(* IEC 61131-3 sources: ATCMcontrol_Engineering/src/TargetBase/Libs/ATCM_XMLfile, 11 files *)

(* ---- XMLClose.st ---- *)
(*[[
    UserURL="ATCMfile:XMLClose.htm",
]]*)
FUNCTION XMLClose:DWORD
VAR_INPUT
    XMLhandle : DINT;
END_VAR

inline { STDLIB(XMLClose) }

END_FUNCTION

(* ---- XMLOpen.st ---- *)
(*[[
    UserURL="ATCMfile:XMLOpen.htm",
]]*)
FUNCTION XMLOpen:DWORD
VAR_INPUT
    path : STRING;
    mode : WORD;
END_VAR
VAR_OUTPUT
    XMLhandle : DINT;
END_VAR

inline { STDLIB(XMLOpen) }

END_FUNCTION

(* ---- XMLRead.st ---- *)
(*[[
    UserURL="ATCMfile:XMLRead.htm",
]]*)
FUNCTION XMLRead:DWORD
VAR_INPUT
    XMLhandle : DINT;
    XmlPath : STRING;
    VarName : STRING;
END_VAR

inline { STDLIB(XMLRead) }

END_FUNCTION

(* ---- XMLReadAttribute.st ---- *)
(*[[
    UserURL="ATCMfile:XMLReadAttribute.htm",
]]*)
FUNCTION XMLReadAttribute:DWORD
VAR_INPUT
    XMLhandle : DINT;
    XmlPath : STRING;
    XmlAttribName : STRING;
    VarName : STRING;
END_VAR

inline { STDLIB(XMLReadAttribute) }

END_FUNCTION

(* ---- XMLReadAttributeEx.st ---- *)
(*[[
    UserURL="ATCMfile:XMLReadAttributeEx.htm",
]]*)
FUNCTION XMLReadAttributeEx:DWORD
VAR_INPUT
    XMLhandle : DINT;
    XmlPath : STRING;
    XmlAttribName : STRING;
	Mode :    WORD;
    VarName : STRING;
END_VAR

inline { STDLIB(XMLReadAttributeEx) }

END_FUNCTION

(* ---- XMLReadEx.st ---- *)
(*[[
    UserURL="ATCMfile:XMLReadEx.htm",
]]*)
FUNCTION XMLReadEx:DWORD
VAR_INPUT
    XMLhandle : DINT;
    XmlPath : STRING;
	Mode :    WORD;
    VarName : STRING;
END_VAR

inline { STDLIB(XMLReadEx) }

END_FUNCTION

(* ---- XMLRemove.st ---- *)
(*[[
    UserURL="ATCMfile:XMLRemove.htm",
]]*)
FUNCTION XMLRemove:DWORD
VAR_INPUT
    XMLhandle : DINT;
    XmlPath : STRING;
END_VAR

inline { STDLIB(XMLRemove) }

END_FUNCTION

(* ---- XMLRemoveAttribute.st ---- *)
(*[[
    UserURL="ATCMfile:XMLRemoveAttribute.htm",
]]*)
FUNCTION XMLRemoveAttribute:DWORD
VAR_INPUT
    XMLhandle : DINT;
    XmlPath : STRING;
    XmlAttribName : STRING;
END_VAR

inline { STDLIB(XMLRemoveAttribute) }

END_FUNCTION

(* ---- XMLSave.st ---- *)
(*[[
    UserURL="ATCMfile:XMLSave.htm",
]]*)
FUNCTION XMLSave:DWORD
VAR_INPUT
    XMLhandle : DINT;
END_VAR

inline { STDLIB(XMLSave) }

END_FUNCTION

(* ---- XMLWrite.st ---- *)
(*[[
    UserURL="ATCMfile:XMLWrite.htm",
]]*)
FUNCTION XMLWrite:DWORD
VAR_INPUT
    XMLhandle : DINT;
    XmlPath : STRING;
    Mode    : INT;
    VarName : STRING;
END_VAR

inline { STDLIB(XMLWrite) }

END_FUNCTION

(* ---- XMLWriteAttribute.st ---- *)
(*[[
    UserURL="ATCMfile:XMLWriteAttribute.htm",
]]*)
FUNCTION XMLWriteAttribute:DWORD
VAR_INPUT
    XMLhandle : DINT;
    XmlPath : STRING;
    XmlAttribName : STRING;
    Mode    : INT;
    VarName : STRING;
END_VAR

inline { STDLIB(XMLWriteAttribute) }

END_FUNCTION
